FUNCTION_BLOCK IEEE1451_ACTUATOR
  {SET_ATTRIBUTE(OpcUa, SERVICE)}
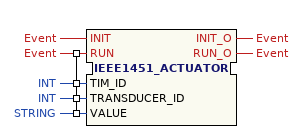
  EVENT_INPUT
    INIT; (* FB Initialization *)
    RUN WITH TIM_ID, TRANSDUCER_ID, VALUE; (* Write Actuator Request *)
  END_EVENT
  EVENT_OUTPUT
    INIT_O; (* Initialization Confirm *)
    RUN_O; (* Write Request Confirm *)
  END_EVENT
  VAR_INPUT
    TIM_ID : INT; (* TIM Identification *)
    TRANSDUCER_ID : INT; (* Transducer Identification *)
    VALUE : STRING; (* Output Data *)
  END_VAR
END_FUNCTION_BLOCK
